{attribute 'GeneratedUsingTerminal: EL4011-0000-0016'}
{attribute addProperty BoxType "EL4011-0000-0016"}
{attribute addProperty Id "AO_OutputsAT %Q*AO_Outputs_BA7EBB7C2WcStateAT %I*WcState_0B2B16F91InfoDataAT %I*InfoData_94A18F5E2"}
{attribute addProperty CRC "3372769853"}
{attribute addProperty Size "5"}
TYPE EL4011_C908623D EXTENDS EtcSlaveTerminalBase_947E5A46 :
STRUCT
	{attribute addProperty Name "AO_Outputs"}
	AO_Outputs : AO_Outputs_BA7EBB7C;
	{attribute addProperty Name "WcState"}
	WcState : WcState_0B2B16F9;
	{attribute addProperty Name "InfoData"}
	InfoData : InfoData_94A18F5E;
END_STRUCT
END_TYPE

(* stored: Version 1.2.0.0, ProductVersion 3.1.4024.9
   DUT EL4011_C908623D: Id {3fa7dad4-602f-4ba5-a7df-2aad0481d763} *)
